TYPE EcSoeWrite_CMD_typ :
	STRUCT
		Enable	: BOOL ;
	END_STRUCT
END_TYPE

(* stored: Version 1.1.0.1, ProductVersion 3.1.4024.3
   DUT EcSoeWrite_CMD_typ: Id {e9e70584-068b-065d-1dd1-dcc8701bacd6} *)
